PROGRAM MAIN
VAR
	// Objects
	SimulatedIO : FB_SimulatedIO;
	Pump : FB_Pump;
	PumpController : FB_PumpController := (nTargetPressure := TARGET_PRESSURE, nMaximumPressure := MAXIMUM_PRESSURE,
		nMinimumPressure := MINIMUM_PRESSURE, nInitialPressure := Pump.nPressure);
	
	// Variables for Graph
	aGraphPoints : ARRAY[1..1, 1..1000] OF ST_Point;
	nPollDelay : UINT := 10; 
	nCurrentPoint : INT := 1;
	nPollCount : UINT := 0;
	
	// Main Loop Variables
	bTurnPumpControllerOn : BOOL := FALSE;
	bPumpState : BOOL := FALSE;
	bEmergencyStopPump : BOOL := FALSE;
	sState : STRING(20) := 'IDLE';
	bManualPump : BOOL := FALSE;
	bManualRelease : BOOL := FALSE;
END_VAR
VAR CONSTANT
	MAXIMUM_PRESSURE : USINT := 10;
	MINIMUM_PRESSURE : USINT := 8;
	TARGET_PRESSURE : USINT := 9;
END_VAR

IF GVL_VAR.bReset THEN
	bEmergencyStopPump := FALSE;
	GVL_VAR.bLeakDetected := FALSE;
	GVL_VAR.bBrokenPump := FALSE;
	GVL_VAR.bReset := FALSE;
	bTurnPumpControllerOn := FALSE;
	bManualPump := FALSE;
	bManualRelease := FALSE;
ELSIF NOT bEmergencyStopPump AND NOT GVL_VAR.bLeakDetected AND NOT GVL_VAR.bBrokenPump THEN // All Systems Normal
	sState := 'IDLING';
	IF bTurnPumpControllerOn THEN
		PumpController.Run(bTurnPumpControllerOn);
		bPumpState := PumpController.bPumpState;
		Pump.SetRelay(bPumpState);
		IF bPumpState THEN
			sState := 'PUMPING';
		END_IF
	ELSIF bManualRelease THEN
		sState := 'M_RELEASE';
		Pump.SetValve(TRUE);
		Pump.SetRelay(FALSE);
	ELSIF bManualPump THEN
		sState := 'M_PUMPING';
		Pump.SetRelay(TRUE);
		Pump.SetValve(FALSE);
	ELSE
		PUMP.SetRelay(FALSE);
		PUMP.SetValve(FALSE);
	END_IF
	
ELSE // Some Error! 
	IF GVL_VAR.bBrokenPump THEN
		sState := 'PUMP_BROKE';
	ELSIF bEmergencyStopPump THEN
		sState := 'E_STOPPED';
	ELSIF GVL_Var.bLeakDetected THEN
		sState := 'LEAK!';
	END_IF
	Pump.SetRelay(FALSE);
	bTurnPumpControllerOn := FALSE;
END_IF

// Save pressure data for graph
IF nCurrentPoint > 1000 THEN
	nCurrentPoint := 2;
	nPollCount := 2;
ELSIF nPollCount > 9 THEN
	aGraphPoints[1, nCurrentPoint].x := nCurrentPoint;
	aGraphPoints[1, nCurrentPoint].y := Pump.nPressure;
	nPollCount := 0;
	nCurrentPoint := 1 + nCurrentPoint;
ELSE
	nPollCount := nPollCount + 1;
END_IF

Pump();
// Simulate I/O
SimulatedIO();

END_PROGRAM

(* stored: Version 1.1.0.1, ProductVersion 3.1.4024.12
   POU MAIN: Id {4806e156-ebbf-4070-8291-7b3f5e6f80bf}, SpecialFunc None *)
